{attribute 'GeneratedUsingTerminal: EK1122-0000-0018'}
{attribute addProperty BoxType "EK1122-0000-0018"}
{attribute addProperty Id "Beckhoff_EL30xxsub_EK1100EK1100_AB5A94672"}
{attribute addProperty CRC "2210396417"}
{attribute addProperty Size "2"}
TYPE Beckhoff_EL30xxEK1122_83BFF901 EXTENDS EK1122_AB5A9467 :
STRUCT
	{attribute addProperty Name "Beckhoff_EL30xxsub_EK1100"}
	{attribute addProperty PreviousPort "Beckhoff EL30xxEK1122 : D"}
	Beckhoff_EL30xxsub_EK1100 : EK1100_AB5A9467;
END_STRUCT
END_TYPE

(* stored: Version 1.2.0.0, ProductVersion 3.1.4024.9
   DUT Beckhoff_EL30xxEK1122_83BFF901: Id {279ba06c-ce18-4292-b6fc-cb18ee2ae9c3} *)
